RoboDK station: kr30 cnc template half inch flat end mill - paulina.rdk

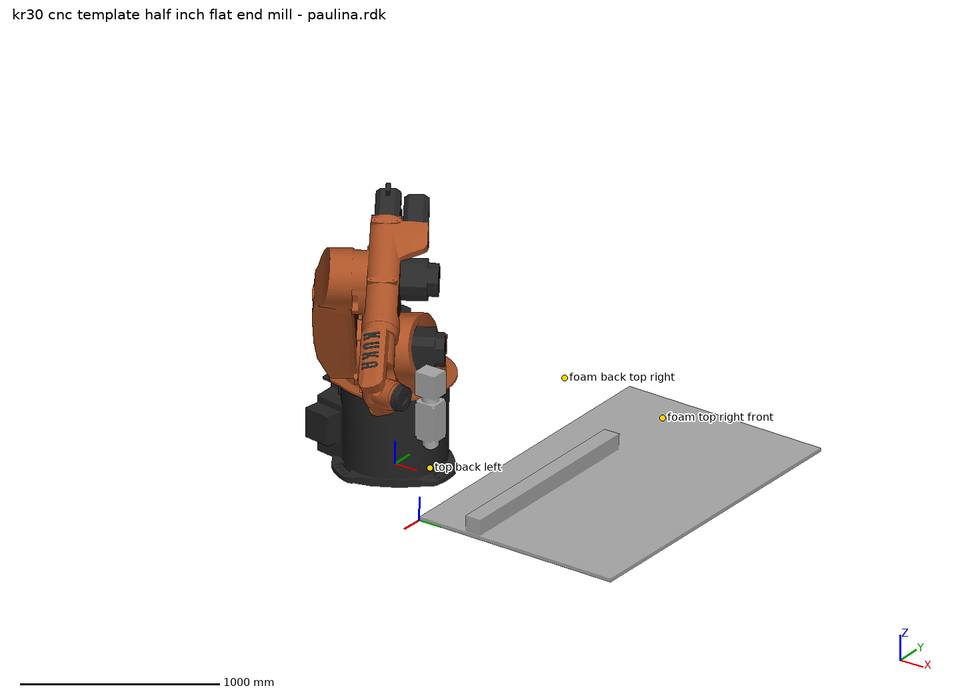
[picture v0: the station drawn from its stored meshes, robots at their saved joint values, targets as dots, program paths as lines]
Station kr30 cnc template half inch flat end mill - paulina. Poses are relative to the parent item; angles as X-Y-Z fixed-axis rotations.
  - frame KUKA KR 30 HA Base at (0, 0, 0) mm
    - robot KUKA KR 30 HA: 6 axes, payload 30 kg, reach 2033 mm, repeatability 0.05 mm, weight 665 kg
        modified DH rows (alpha deg, a mm, theta deg, d mm): 0, 0, 0, 815; -90, 350, 0, 0; 0, 850, -90, 0; -90, 145, 0, 820; 90, 0, 0, 0; -90, 0, 180, 170
        joint limits [-185, -135, -120, -350, -119, -350] to [185, 35, 158, 350, 119, 350]; home [0, -90, 90, 0, 0, 0]; saved at [58.171, -50.232, 76.73, 74.515, -61.834, -59.599]
      - tool rc90 spindle mm, TCP at (337.31, -2.2, 160.57) mm, size 110 x 421.3 x 118 mm, geometry from rc90 spindle mm.stl
    - frame Tabletop at (921.82, -1104.91, 385) mm, rotated rx -0.93 ry -0.21 rz -89.9 deg
      - object tabletop CHECK HEIGHT at (-1839.9, 0, 0) mm, size 1839.9 x 1168.4 x 19 mm, geometry from kr30 tabletop mm.stl
      - object kr30 pipe jig base at (-1220, -610.6, 0) mm, size 1217.6 x 88.9 x 88.9 mm, geometry from kr30 pipe jig base.stl
    - target foam back top right (Cartesian target) at (1197.65, -230.62, 906.79) mm, rotated rx -15.53 ry 90 rz -15.53 deg; joints [14.757, -102.447, 141.256, 22.791, -41.102, -17.568] of KUKA KR 30 HA
    - target foam top right front (Cartesian target) at (1797.45, -230.62, 850.68) mm, rotated rx -15.58 ry 90 rz -15.58 deg; joints [8.85, -62.405, 99.608, 14.434, -38.093, -11.451] of KUKA KR 30 HA
    - target top back left (Cartesian target) at (1223.08, -1440.01, 894.96) mm, rotated rx 58.97 ry 90 rz 58.97 deg; joints [58.171, -50.232, 76.73, 74.515, -61.834, -59.599] of KUKA KR 30 HA
